{attribute 'GeneratedUsingTerminal: EJ4002-0000-0017'}
{attribute addProperty BoxType "EJ4002-0000-0017"}
{attribute addProperty Id "AO_Outputs_Channel_1AT %Q*AO_Outputs_Channel_BA7EBB7C2AO_Outputs_Channel_2AT %Q*AO_Outputs_Channel_BA7EBB7C2WcStateAT %I*WcState_0B2B16F91InfoDataAT %I*InfoData_94A18F5E2"}
{attribute addProperty CRC "3996573741"}
{attribute addProperty Size "7"}
TYPE EJ4002_EE36E02D EXTENDS EtcSlaveTerminalBase_947E5A46 :
STRUCT
	{attribute addProperty Name "AO_Outputs_Channel_1"}
	AO_Outputs_Channel_1 : AO_Outputs_Channel_BA7EBB7C;
	{attribute addProperty Name "AO_Outputs_Channel_2"}
	AO_Outputs_Channel_2 : AO_Outputs_Channel_BA7EBB7C;
	{attribute addProperty Name "WcState"}
	WcState : WcState_0B2B16F9;
	{attribute addProperty Name "InfoData"}
	InfoData : InfoData_94A18F5E;
END_STRUCT
END_TYPE

(* stored: Version 1.2.0.0, ProductVersion 3.1.4024.9
   DUT EJ4002_EE36E02D: Id {30bd6b70-4228-4a64-8055-ac62cd134578} *)
